{attribute 'qualified_only'}
VAR_GLOBAL
	Communication		:ModbusRtuMasterV2_PcCOM;
END_VAR

(* stored: Version 1.1.0.1
   GVL GVL: Id {d358711c-d4bb-4176-9fa5-bdda4bc55262} *)
